{attribute 'GeneratedUsingTerminal: EK1100-0000-0018'}
{attribute addProperty BoxType "EK1100-0000-0018"}
{attribute addProperty Id "R4_A2_EC_EK1122R4_A2_EC_EK1122_254454A1269R4_A3_DI_EL1809EL1809_32157CFD20R4_A4_DI_EL1809EL1809_32157CFD20R4_A5_DI_EL1809EL1809_32157CFD20R4_A6_DI_EL1809EL1809_32157CFD20R4_A7_DI_EL1809EL1809_32157CFD20R4_EndTerminal_EL9011EL9011_D65D3D320"}
{attribute addProperty CRC "1184965772"}
{attribute addProperty Size "369"}
{attribute addProperty Name "R4 (EK1100)"}
TYPE R4_EK1100_46A1248C EXTENDS EK1100_1FC0878B :
STRUCT
	{attribute addProperty Name "R4_A2_EC (EK1122)"}
	{attribute addProperty PreviousPort "R4 (EK1100) : B"}
	{attribute addProperty SyncUnit "default"}
	R4_A2_EC_EK1122 : R4_A2_EC_EK1122_254454A1;
	{attribute addProperty Name "R4_A3_DI (EL1809)"}
	{attribute addProperty PreviousPort "R4_A2_EC (EK1122) : C"}
	{attribute addProperty SyncUnit "default"}
	R4_A3_DI_EL1809 : EL1809_32157CFD;
	{attribute addProperty Name "R4_A4_DI (EL1809)"}
	{attribute addProperty PreviousPort "R4_A3_DI (EL1809) : B"}
	{attribute addProperty SyncUnit "default"}
	R4_A4_DI_EL1809 : EL1809_32157CFD;
	{attribute addProperty Name "R4_A5_DI (EL1809)"}
	{attribute addProperty PreviousPort "R4_A4_DI (EL1809) : B"}
	{attribute addProperty SyncUnit "default"}
	R4_A5_DI_EL1809 : EL1809_32157CFD;
	{attribute addProperty Name "R4_A6_DI (EL1809)"}
	{attribute addProperty PreviousPort "R4_A5_DI (EL1809) : B"}
	{attribute addProperty SyncUnit "default"}
	R4_A6_DI_EL1809 : EL1809_32157CFD;
	{attribute addProperty Name "R4_A7_DI (EL1809)"}
	{attribute addProperty PreviousPort "R4_A6_DI (EL1809) : B"}
	{attribute addProperty SyncUnit "default"}
	R4_A7_DI_EL1809 : EL1809_32157CFD;
	{attribute addProperty Name "R4_EndTerminal (EL9011)"}
	{attribute addProperty PreviousPort "R4_A7_DI (EL1809) : B"}
	{attribute addProperty SyncUnit "default"}
	R4_EndTerminal_EL9011 : EL9011_D65D3D32;
END_STRUCT
END_TYPE

(* stored: Version 1.2.0.0, ProductVersion 3.1.4024.11
   DUT R4_EK1100_46A1248C: Id {2f121970-17ad-0d7a-2d8e-7e5b949413f8} *)
